// TIA Portal V21 export
FUNCTION_BLOCK "FB110"   // FB110, LAD
TITLE = FB110
{ S7_Optimized_Access := 'FALSE' }
// Step Delay for Delay in Valves
// stored: AutoNumber false, SetENOAutomatically false
   VAR_INPUT
      Enable : Bool;
      Running : Bool;
      SecPulse : Bool;
      AlwaysOn : Bool;
      "NoOf StepsSv" : Int;
      StepTimeSv : Array[0..18] of Int;
   END_VAR
   VAR_OUTPUT
      StepTimePv : DInt;
      Done : Bool;
   END_VAR
   VAR_IN_OUT
      Selected : Bool;
      StepStarted : Bool;
      SelectionRe : Bool;
      StepStartedRe : Bool;
      NextStepTrigger : Bool;
      "Noof StepsPv" : Int;
      StepTime : Int;
      Temp : Int;
   END_VAR
   VAR
      TimerInstance { S7_SetPoint := 'True'} : "FB101";
   END_VAR
   // StepTimeSv[1..10] := 10;
   VAR_TEMP   // added for the SCL form of the ladder/FBD networks
      _w1 : Bool;
      _w2 : Bool;
   END_VAR
BEGIN

REGION Network 1: Selected
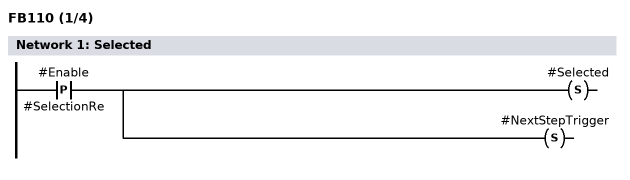
   RUNG wire#powerrail
      P_Contact(operand := #Enable, bit := #SelectionRe)
      wire#w1
      S_Coil( #Selected )
   END_RUNG
   RUNG wire#w1
      S_Coil( #NextStepTrigger )
   END_RUNG
   // the same network as SCL:
   #_w1 := #Enable AND NOT #SelectionRe;   // rising edge of #Enable
   #SelectionRe := #Enable;
   IF #_w1 THEN
       #Selected := TRUE;
       #NextStepTrigger := TRUE;
   END_IF;
END_REGION

REGION Network 2: Step Time
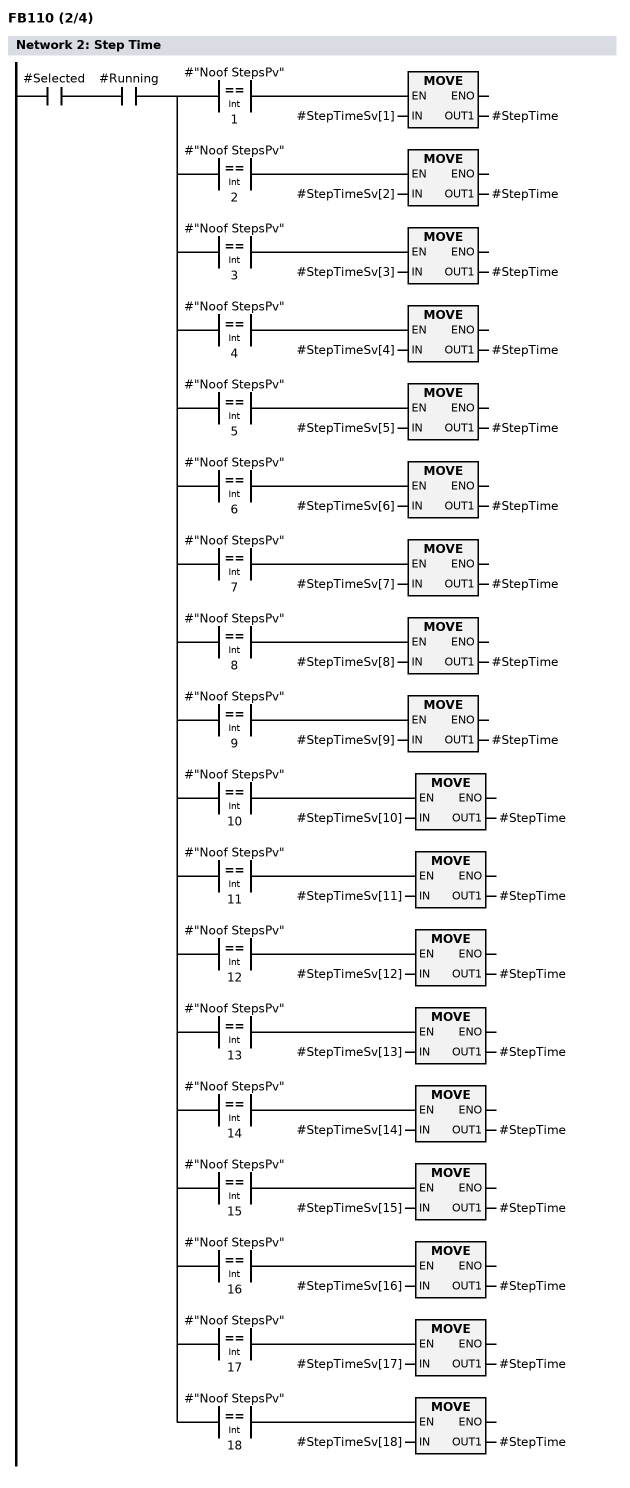
   RUNG wire#powerrail
      Contact( #Selected )
      Contact( #Running )
      wire#w1
      { S7_Templates := "SrcType := Int" } EQ_Contact(in1 := #"Noof StepsPv", in2 := 1)
      { S7_GenerateENO := "TRUE" } Move(in := #StepTimeSv[1], out1 => #StepTime)
   END_RUNG
   RUNG wire#w1
      { S7_Templates := "SrcType := Int" } EQ_Contact(in1 := #"Noof StepsPv", in2 := 2)
      { S7_GenerateENO := "TRUE" } Move(in := #StepTimeSv[2], out1 => #StepTime)
   END_RUNG
   RUNG wire#w1
      { S7_Templates := "SrcType := Int" } EQ_Contact(in1 := #"Noof StepsPv", in2 := 3)
      { S7_GenerateENO := "TRUE" } Move(in := #StepTimeSv[3], out1 => #StepTime)
   END_RUNG
   RUNG wire#w1
      { S7_Templates := "SrcType := Int" } EQ_Contact(in1 := #"Noof StepsPv", in2 := 4)
      { S7_GenerateENO := "TRUE" } Move(in := #StepTimeSv[4], out1 => #StepTime)
   END_RUNG
   RUNG wire#w1
      { S7_Templates := "SrcType := Int" } EQ_Contact(in1 := #"Noof StepsPv", in2 := 5)
      { S7_GenerateENO := "TRUE" } Move(in := #StepTimeSv[5], out1 => #StepTime)
   END_RUNG
   RUNG wire#w1
      { S7_Templates := "SrcType := Int" } EQ_Contact(in1 := #"Noof StepsPv", in2 := 6)
      { S7_GenerateENO := "TRUE" } Move(in := #StepTimeSv[6], out1 => #StepTime)
   END_RUNG
   RUNG wire#w1
      { S7_Templates := "SrcType := Int" } EQ_Contact(in1 := #"Noof StepsPv", in2 := 7)
      { S7_GenerateENO := "TRUE" } Move(in := #StepTimeSv[7], out1 => #StepTime)
   END_RUNG
   RUNG wire#w1
      { S7_Templates := "SrcType := Int" } EQ_Contact(in1 := #"Noof StepsPv", in2 := 8)
      { S7_GenerateENO := "TRUE" } Move(in := #StepTimeSv[8], out1 => #StepTime)
   END_RUNG
   RUNG wire#w1
      { S7_Templates := "SrcType := Int" } EQ_Contact(in1 := #"Noof StepsPv", in2 := 9)
      { S7_GenerateENO := "TRUE" } Move(in := #StepTimeSv[9], out1 => #StepTime)
   END_RUNG
   RUNG wire#w1
      { S7_Templates := "SrcType := Int" } EQ_Contact(in1 := #"Noof StepsPv", in2 := 10)
      { S7_GenerateENO := "TRUE" } Move(in := #StepTimeSv[10], out1 => #StepTime)
   END_RUNG
   RUNG wire#w1
      { S7_Templates := "SrcType := Int" } EQ_Contact(in1 := #"Noof StepsPv", in2 := 11)
      { S7_GenerateENO := "TRUE" } Move(in := #StepTimeSv[11], out1 => #StepTime)
   END_RUNG
   RUNG wire#w1
      { S7_Templates := "SrcType := Int" } EQ_Contact(in1 := #"Noof StepsPv", in2 := 12)
      { S7_GenerateENO := "TRUE" } Move(in := #StepTimeSv[12], out1 => #StepTime)
   END_RUNG
   RUNG wire#w1
      { S7_Templates := "SrcType := Int" } EQ_Contact(in1 := #"Noof StepsPv", in2 := 13)
      { S7_GenerateENO := "TRUE" } Move(in := #StepTimeSv[13], out1 => #StepTime)
   END_RUNG
   RUNG wire#w1
      { S7_Templates := "SrcType := Int" } EQ_Contact(in1 := #"Noof StepsPv", in2 := 14)
      { S7_GenerateENO := "TRUE" } Move(in := #StepTimeSv[14], out1 => #StepTime)
   END_RUNG
   RUNG wire#w1
      { S7_Templates := "SrcType := Int" } EQ_Contact(in1 := #"Noof StepsPv", in2 := 15)
      { S7_GenerateENO := "TRUE" } Move(in := #StepTimeSv[15], out1 => #StepTime)
   END_RUNG
   RUNG wire#w1
      { S7_Templates := "SrcType := Int" } EQ_Contact(in1 := #"Noof StepsPv", in2 := 16)
      { S7_GenerateENO := "TRUE" } Move(in := #StepTimeSv[16], out1 => #StepTime)
   END_RUNG
   RUNG wire#w1
      { S7_Templates := "SrcType := Int" } EQ_Contact(in1 := #"Noof StepsPv", in2 := 17)
      { S7_GenerateENO := "TRUE" } Move(in := #StepTimeSv[17], out1 => #StepTime)
   END_RUNG
   RUNG wire#w1
      { S7_Templates := "SrcType := Int" } EQ_Contact(in1 := #"Noof StepsPv", in2 := 18)
      { S7_GenerateENO := "TRUE" } Move(in := #StepTimeSv[18], out1 => #StepTime)
   END_RUNG
   // the same network as SCL:
   #_w1 := #Selected AND #Running;
   IF #_w1 AND (#"Noof StepsPv" = 1) THEN #StepTime := #StepTimeSv[1]; END_IF;
   IF #_w1 AND (#"Noof StepsPv" = 2) THEN #StepTime := #StepTimeSv[2]; END_IF;
   IF #_w1 AND (#"Noof StepsPv" = 3) THEN #StepTime := #StepTimeSv[3]; END_IF;
   IF #_w1 AND (#"Noof StepsPv" = 4) THEN #StepTime := #StepTimeSv[4]; END_IF;
   IF #_w1 AND (#"Noof StepsPv" = 5) THEN #StepTime := #StepTimeSv[5]; END_IF;
   IF #_w1 AND (#"Noof StepsPv" = 6) THEN #StepTime := #StepTimeSv[6]; END_IF;
   IF #_w1 AND (#"Noof StepsPv" = 7) THEN #StepTime := #StepTimeSv[7]; END_IF;
   IF #_w1 AND (#"Noof StepsPv" = 8) THEN #StepTime := #StepTimeSv[8]; END_IF;
   IF #_w1 AND (#"Noof StepsPv" = 9) THEN #StepTime := #StepTimeSv[9]; END_IF;
   IF #_w1 AND (#"Noof StepsPv" = 10) THEN #StepTime := #StepTimeSv[10]; END_IF;
   IF #_w1 AND (#"Noof StepsPv" = 11) THEN #StepTime := #StepTimeSv[11]; END_IF;
   IF #_w1 AND (#"Noof StepsPv" = 12) THEN #StepTime := #StepTimeSv[12]; END_IF;
   IF #_w1 AND (#"Noof StepsPv" = 13) THEN #StepTime := #StepTimeSv[13]; END_IF;
   IF #_w1 AND (#"Noof StepsPv" = 14) THEN #StepTime := #StepTimeSv[14]; END_IF;
   IF #_w1 AND (#"Noof StepsPv" = 15) THEN #StepTime := #StepTimeSv[15]; END_IF;
   IF #_w1 AND (#"Noof StepsPv" = 16) THEN #StepTime := #StepTimeSv[16]; END_IF;
   IF #_w1 AND (#"Noof StepsPv" = 17) THEN #StepTime := #StepTimeSv[17]; END_IF;
   IF #_w1 AND (#"Noof StepsPv" = 18) THEN #StepTime := #StepTimeSv[18]; END_IF;
END_REGION

REGION Network 3: Step Timer
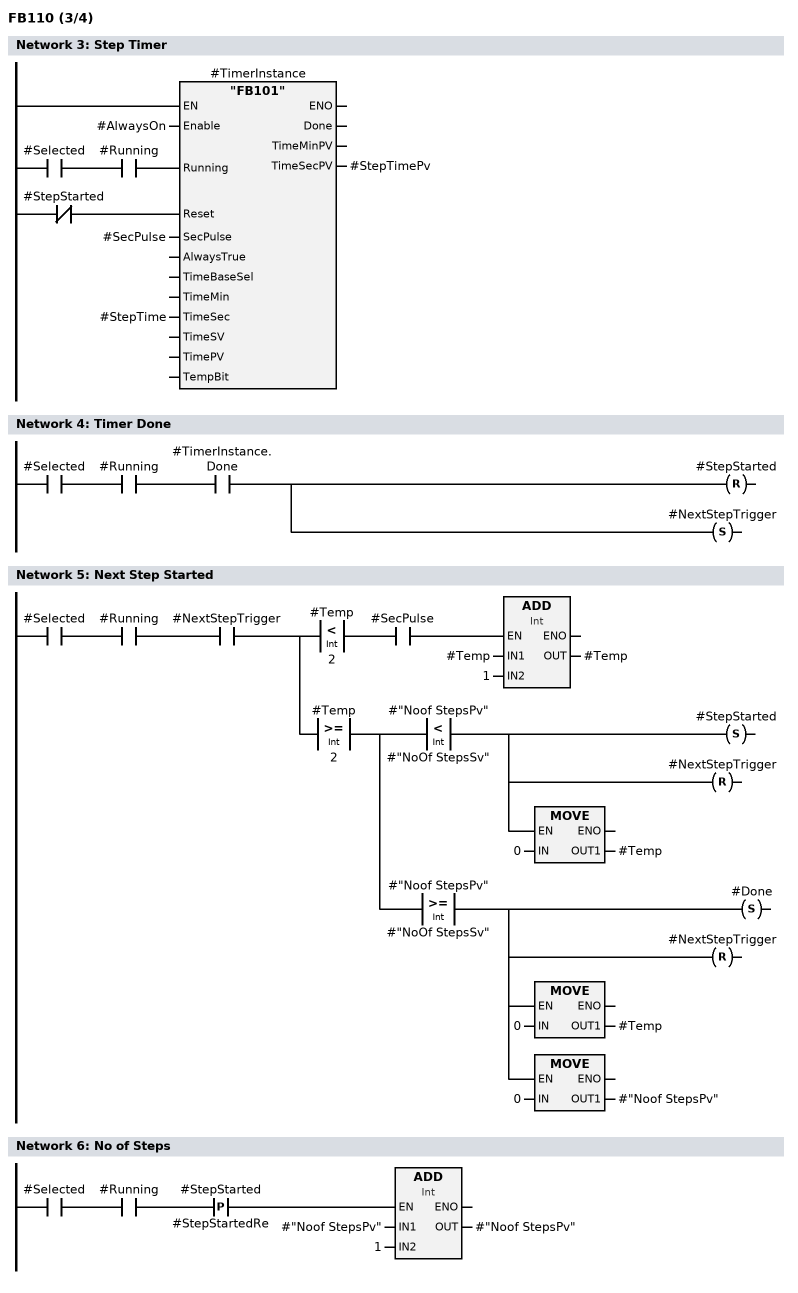
   RUNG wire#powerrail
      #TimerInstance(Running := wire#w1, Reset := wire#w2, Enable := #AlwaysOn, SecPulse := #SecPulse, AlwaysTrue :=, TimeBaseSel :=, TimeMin :=, TimeSec := #StepTime, TimeSV :=, TimePV :=, TempBit :=, Done =>, TimeMinPV =>, TimeSecPV => #StepTimePv)
   END_RUNG
   RUNG wire#powerrail
      Contact( #Selected )
      Contact( #Running )
   END_RUNG wire#w1
   RUNG wire#powerrail
      I_Contact( #StepStarted )
   END_RUNG wire#w2
   // the same network as SCL:
   #TimerInstance(Enable := #AlwaysOn,   // "FB101"
                  Running := #Selected AND #Running,
                  Reset := NOT #StepStarted,
                  SecPulse := #SecPulse,
                  TimeSec := #StepTime,
                  TimeSecPV => #StepTimePv);
END_REGION

REGION Network 4: Timer Done
   RUNG wire#powerrail
      Contact( #Selected )
      Contact( #Running )
      Contact( #TimerInstance.Done )
      wire#w1
      R_Coil( #StepStarted )
   END_RUNG
   RUNG wire#w1
      S_Coil( #NextStepTrigger )
   END_RUNG
   // the same network as SCL:
   IF #Selected AND #Running AND #TimerInstance.Done THEN
       #StepStarted := FALSE;
       #NextStepTrigger := TRUE;
   END_IF;
END_REGION

REGION Network 5: Next Step Started
   RUNG wire#powerrail
      Contact( #Selected )
      Contact( #Running )
      Contact( #NextStepTrigger )
      wire#w1
      { S7_Templates := "SrcType := Int" } LT_Contact(in1 := #Temp, in2 := 2)
      Contact( #SecPulse )
      { S7_Templates := "SrcType := Int"; S7_GenerateENO := "TRUE" } Add(in1 := #Temp, in2 := 1, out => #Temp)
   END_RUNG
   RUNG wire#w1
      { S7_Templates := "SrcType := Int" } GE_Contact(in1 := #Temp, in2 := 2)
      wire#w2
      { S7_Templates := "SrcType := Int" } LT_Contact(in1 := #"Noof StepsPv", in2 := #"NoOf StepsSv")
      wire#w3
      S_Coil( #StepStarted )
   END_RUNG
   RUNG wire#w3
      R_Coil( #NextStepTrigger )
   END_RUNG
   RUNG wire#w3
      { S7_GenerateENO := "TRUE" } Move(in := 0, out1 => #Temp)
   END_RUNG
   RUNG wire#w2
      { S7_Templates := "SrcType := Int" } GE_Contact(in1 := #"Noof StepsPv", in2 := #"NoOf StepsSv")
      wire#w4
      S_Coil( #Done )
   END_RUNG
   RUNG wire#w4
      R_Coil( #NextStepTrigger )
   END_RUNG
   RUNG wire#w4
      { S7_GenerateENO := "TRUE" } Move(in := 0, out1 => #Temp)
   END_RUNG
   RUNG wire#w4
      { S7_GenerateENO := "TRUE" } Move(in := 0, out1 => #"Noof StepsPv")
   END_RUNG
   // the same network as SCL:
   #_w1 := #Selected AND #Running AND #NextStepTrigger;
   IF #_w1 AND (#Temp < 2) AND #SecPulse THEN #Temp := #Temp + 1; END_IF;
   #_w2 := #_w1 AND (#Temp >= 2);
   IF #_w2 AND (#"Noof StepsPv" < #"NoOf StepsSv") THEN
       #StepStarted := TRUE;
       #NextStepTrigger := FALSE;
       #Temp := 0;
   END_IF;
   IF #_w2 AND (#"Noof StepsPv" >= #"NoOf StepsSv") THEN
       #Done := TRUE;
       #NextStepTrigger := FALSE;
       #Temp := 0;
       #"Noof StepsPv" := 0;
   END_IF;
END_REGION

REGION Network 6: No of Steps
   RUNG wire#powerrail
      Contact( #Selected )
      Contact( #Running )
      P_Contact(operand := #StepStarted, bit := #StepStartedRe)
      { S7_Templates := "SrcType := Int"; S7_GenerateENO := "TRUE" } Add(in1 := #"Noof StepsPv", in2 := 1, out => #"Noof StepsPv")
   END_RUNG
   // the same network as SCL:
   #_w1 := #Selected AND #Running AND #StepStarted AND NOT #StepStartedRe;   // rising edge of #StepStarted
   #StepStartedRe := #StepStarted;
   IF #_w1 THEN #"Noof StepsPv" := #"Noof StepsPv" + 1; END_IF;
END_REGION

REGION Network 7: Reset
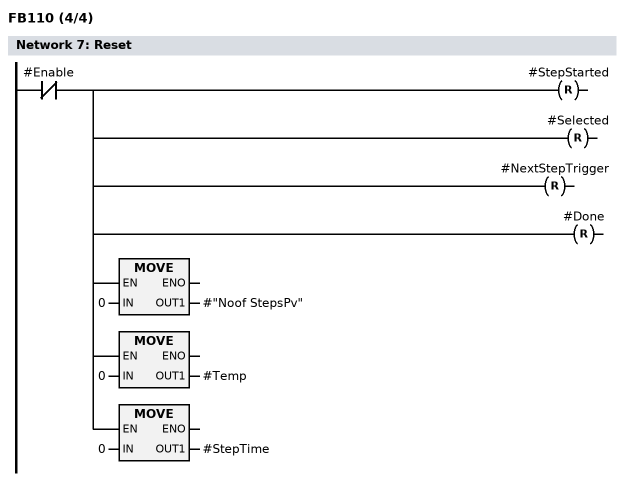
   RUNG wire#powerrail
      I_Contact( #Enable )
      wire#w1
      R_Coil( #StepStarted )
   END_RUNG
   RUNG wire#w1
      R_Coil( #Selected )
   END_RUNG
   RUNG wire#w1
      R_Coil( #NextStepTrigger )
   END_RUNG
   RUNG wire#w1
      R_Coil( #Done )
   END_RUNG
   RUNG wire#w1
      { S7_GenerateENO := "TRUE" } Move(in := 0, out1 => #"Noof StepsPv")
   END_RUNG
   RUNG wire#w1
      { S7_GenerateENO := "TRUE" } Move(in := 0, out1 => #Temp)
   END_RUNG
   RUNG wire#w1
      { S7_GenerateENO := "TRUE" } Move(in := 0, out1 => #StepTime)
   END_RUNG
   // the same network as SCL:
   IF NOT #Enable THEN
       #StepStarted := FALSE;
       #Selected := FALSE;
       #NextStepTrigger := FALSE;
       #Done := FALSE;
       #"Noof StepsPv" := 0;
       #Temp := 0;
       #StepTime := 0;
   END_IF;
END_REGION
END_FUNCTION_BLOCK
